PROGRAM ClangsonicUSCtrl
VAR

END_VAR
VAR // added by the converter: edge detectors and wires of the graphical bodies
    _w1, _w2, _w3, _w4, _w5, _w6, _w7, _w8, _w9, _w10, _w11, _w12, _w13, _w14, _w15, _w16, _w17, _w18 : INT;
END_VAR

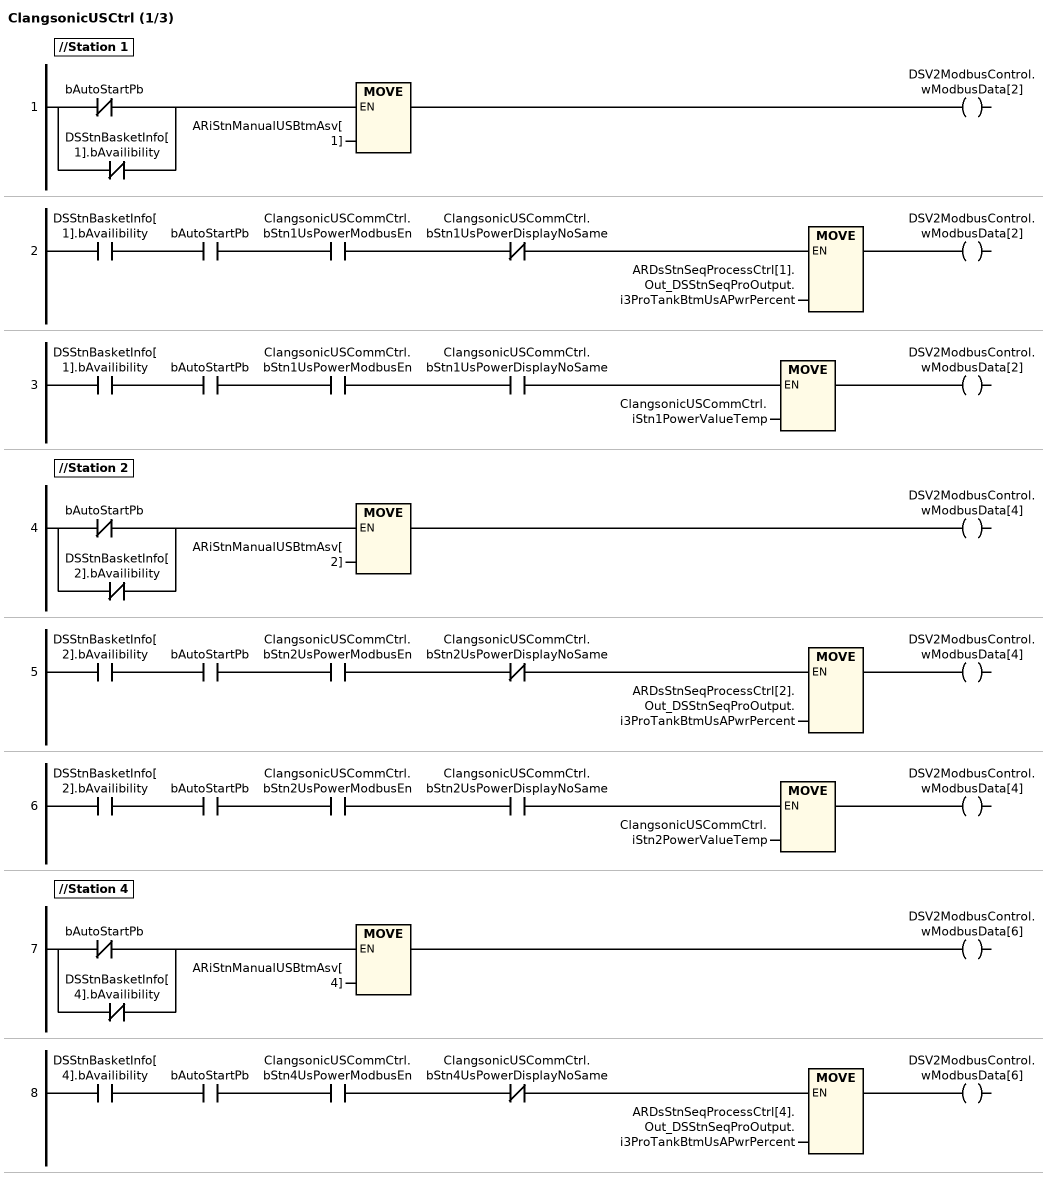
// NETWORK 1
// label: //Station 1
IF NOT bAutoStartPb OR NOT DSStnBasketInfo[1].bAvailibility THEN _w1 := ARiStnManualUSBtmAsv[1]; END_IF
DSV2ModbusControl.wModbusData[2] := _w1;

// NETWORK 2
IF DSStnBasketInfo[1].bAvailibility AND bAutoStartPb AND ClangsonicUSCommCtrl.bStn1UsPowerModbusEn AND NOT ClangsonicUSCommCtrl.bStn1UsPowerDisplayNoSame THEN
    _w2 := ARDsStnSeqProcessCtrl[1].Out_DSStnSeqProOutput.i3ProTankBtmUsAPwrPercent;
END_IF
DSV2ModbusControl.wModbusData[2] := _w2;

// NETWORK 3
IF DSStnBasketInfo[1].bAvailibility AND bAutoStartPb AND ClangsonicUSCommCtrl.bStn1UsPowerModbusEn AND ClangsonicUSCommCtrl.bStn1UsPowerDisplayNoSame THEN
    _w3 := ClangsonicUSCommCtrl.iStn1PowerValueTemp;
END_IF
DSV2ModbusControl.wModbusData[2] := _w3;

// NETWORK 4
// label: //Station 2
IF NOT bAutoStartPb OR NOT DSStnBasketInfo[2].bAvailibility THEN _w4 := ARiStnManualUSBtmAsv[2]; END_IF
DSV2ModbusControl.wModbusData[4] := _w4;

// NETWORK 5
IF DSStnBasketInfo[2].bAvailibility AND bAutoStartPb AND ClangsonicUSCommCtrl.bStn2UsPowerModbusEn AND NOT ClangsonicUSCommCtrl.bStn2UsPowerDisplayNoSame THEN
    _w5 := ARDsStnSeqProcessCtrl[2].Out_DSStnSeqProOutput.i3ProTankBtmUsAPwrPercent;
END_IF
DSV2ModbusControl.wModbusData[4] := _w5;

// NETWORK 6
IF DSStnBasketInfo[2].bAvailibility AND bAutoStartPb AND ClangsonicUSCommCtrl.bStn2UsPowerModbusEn AND ClangsonicUSCommCtrl.bStn2UsPowerDisplayNoSame THEN
    _w6 := ClangsonicUSCommCtrl.iStn2PowerValueTemp;
END_IF
DSV2ModbusControl.wModbusData[4] := _w6;

// NETWORK 7
// label: //Station 4
IF NOT bAutoStartPb OR NOT DSStnBasketInfo[4].bAvailibility THEN _w7 := ARiStnManualUSBtmAsv[4]; END_IF
DSV2ModbusControl.wModbusData[6] := _w7;

// NETWORK 8
IF DSStnBasketInfo[4].bAvailibility AND bAutoStartPb AND ClangsonicUSCommCtrl.bStn4UsPowerModbusEn AND NOT ClangsonicUSCommCtrl.bStn4UsPowerDisplayNoSame THEN
    _w8 := ARDsStnSeqProcessCtrl[4].Out_DSStnSeqProOutput.i3ProTankBtmUsAPwrPercent;
END_IF
DSV2ModbusControl.wModbusData[6] := _w8;

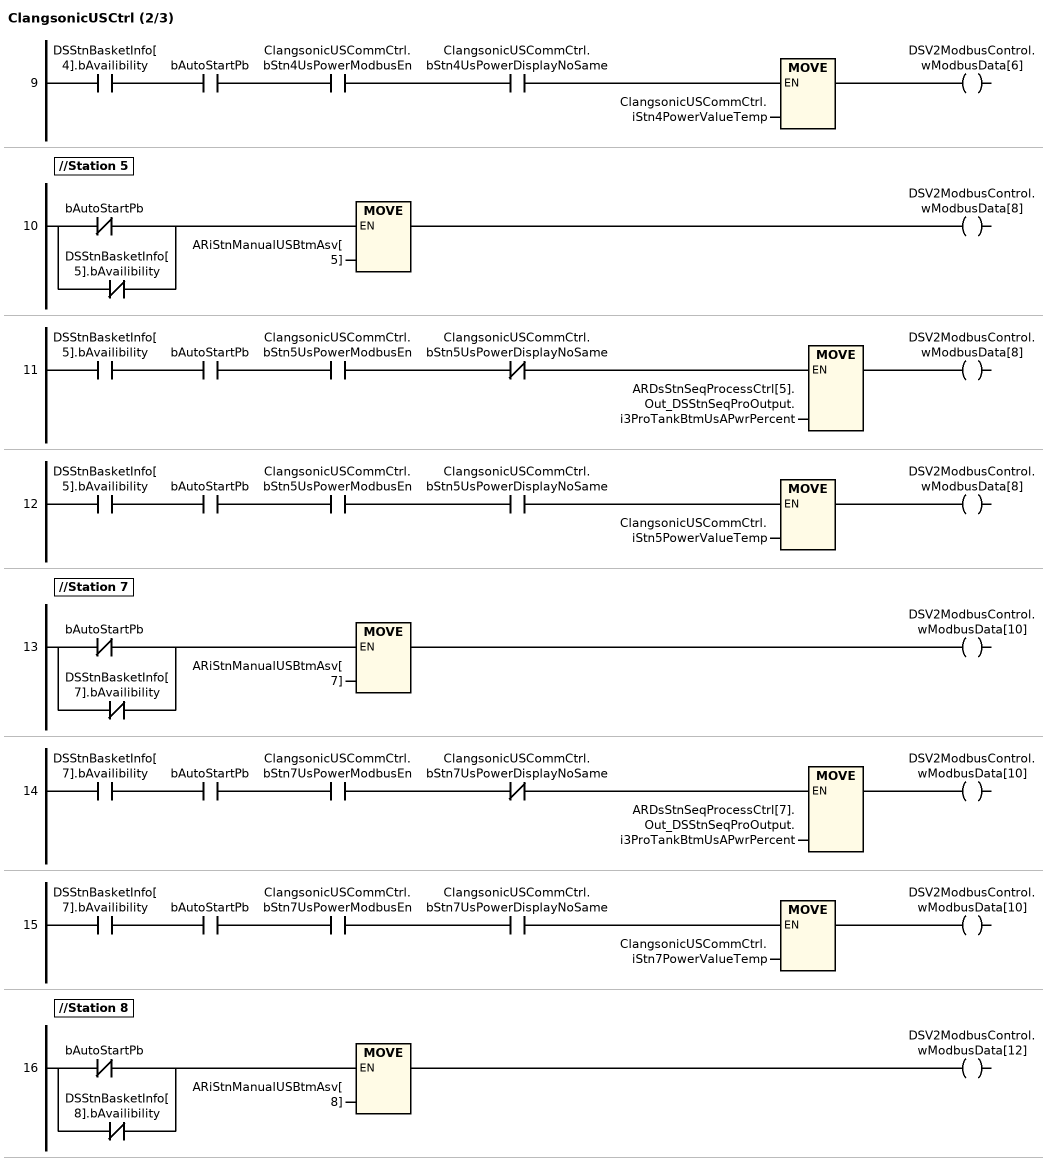
// NETWORK 9
IF DSStnBasketInfo[4].bAvailibility AND bAutoStartPb AND ClangsonicUSCommCtrl.bStn4UsPowerModbusEn AND ClangsonicUSCommCtrl.bStn4UsPowerDisplayNoSame THEN
    _w9 := ClangsonicUSCommCtrl.iStn4PowerValueTemp;
END_IF
DSV2ModbusControl.wModbusData[6] := _w9;

// NETWORK 10
// label: //Station 5
IF NOT bAutoStartPb OR NOT DSStnBasketInfo[5].bAvailibility THEN _w10 := ARiStnManualUSBtmAsv[5]; END_IF
DSV2ModbusControl.wModbusData[8] := _w10;

// NETWORK 11
IF DSStnBasketInfo[5].bAvailibility AND bAutoStartPb AND ClangsonicUSCommCtrl.bStn5UsPowerModbusEn AND NOT ClangsonicUSCommCtrl.bStn5UsPowerDisplayNoSame THEN
    _w11 := ARDsStnSeqProcessCtrl[5].Out_DSStnSeqProOutput.i3ProTankBtmUsAPwrPercent;
END_IF
DSV2ModbusControl.wModbusData[8] := _w11;

// NETWORK 12
IF DSStnBasketInfo[5].bAvailibility AND bAutoStartPb AND ClangsonicUSCommCtrl.bStn5UsPowerModbusEn AND ClangsonicUSCommCtrl.bStn5UsPowerDisplayNoSame THEN
    _w12 := ClangsonicUSCommCtrl.iStn5PowerValueTemp;
END_IF
DSV2ModbusControl.wModbusData[8] := _w12;

// NETWORK 13
// label: //Station 7
IF NOT bAutoStartPb OR NOT DSStnBasketInfo[7].bAvailibility THEN _w13 := ARiStnManualUSBtmAsv[7]; END_IF
DSV2ModbusControl.wModbusData[10] := _w13;

// NETWORK 14
IF DSStnBasketInfo[7].bAvailibility AND bAutoStartPb AND ClangsonicUSCommCtrl.bStn7UsPowerModbusEn AND NOT ClangsonicUSCommCtrl.bStn7UsPowerDisplayNoSame THEN
    _w14 := ARDsStnSeqProcessCtrl[7].Out_DSStnSeqProOutput.i3ProTankBtmUsAPwrPercent;
END_IF
DSV2ModbusControl.wModbusData[10] := _w14;

// NETWORK 15
IF DSStnBasketInfo[7].bAvailibility AND bAutoStartPb AND ClangsonicUSCommCtrl.bStn7UsPowerModbusEn AND ClangsonicUSCommCtrl.bStn7UsPowerDisplayNoSame THEN
    _w15 := ClangsonicUSCommCtrl.iStn7PowerValueTemp;
END_IF
DSV2ModbusControl.wModbusData[10] := _w15;

// NETWORK 16
// label: //Station 8
IF NOT bAutoStartPb OR NOT DSStnBasketInfo[8].bAvailibility THEN _w16 := ARiStnManualUSBtmAsv[8]; END_IF
DSV2ModbusControl.wModbusData[12] := _w16;

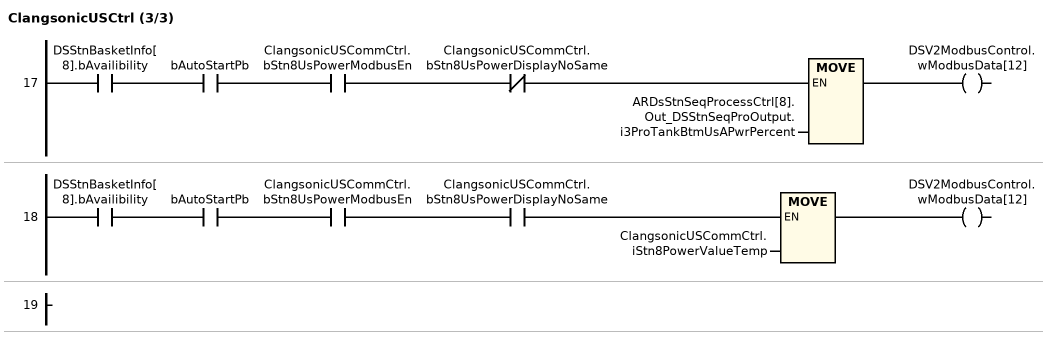
// NETWORK 17
IF DSStnBasketInfo[8].bAvailibility AND bAutoStartPb AND ClangsonicUSCommCtrl.bStn8UsPowerModbusEn AND NOT ClangsonicUSCommCtrl.bStn8UsPowerDisplayNoSame THEN
    _w17 := ARDsStnSeqProcessCtrl[8].Out_DSStnSeqProOutput.i3ProTankBtmUsAPwrPercent;
END_IF
DSV2ModbusControl.wModbusData[12] := _w17;

// NETWORK 18
IF DSStnBasketInfo[8].bAvailibility AND bAutoStartPb AND ClangsonicUSCommCtrl.bStn8UsPowerModbusEn AND ClangsonicUSCommCtrl.bStn8UsPowerDisplayNoSame THEN
    _w18 := ClangsonicUSCommCtrl.iStn8PowerValueTemp;
END_IF
DSV2ModbusControl.wModbusData[12] := _w18;

// NETWORK 19

END_PROGRAM

(* stored: Version 1.1.0.1, ProductVersion 3.1.4024.12
   POU ClangsonicUSCtrl: Id {2b268933-10db-4628-bec5-73a8f625ed67}, SpecialFunc None *)
